KUKA KRL data list: SOLVE_HANOI.DAT

&ACCESS RVO
&REL 66
&PARAM TEMPLATE = C:\KRC\Roboter\Template\ExpertVorgabe
&PARAM EDITMASK = *
DEFDAT  SOLVE_HANOI
DECL INT I=1
DECL GLOBAL INT HANOI_DISK_COUNT=3
; Calculate REQUIRED_MOVES = 2^HANOI_DISK_COUNT - 1 (does KRL have exponents?)
DECL INT REQUIRED_MOVES=7
DECL INT MOVE_ARRAY[7,2]
DECL INT DISK_COUNTS[3]

; Remember if we come from HOME
DECL BOOL FirstMove=FALSE

; Tool Definitions
DECL GLOBAL FRAME DiskTool={x 0.0,y 0.0,z 150.0,a 0.5,b -90.5,c 0.0}

; Following are placeholders
; Info about the disk in
DECL GLOBAL REAL DISK_THICKNESS=36.65
DECL GLOBAL REAL DISK_PICKUP_OFFSET=-17

; Pick-up zone X offset
DECL GLOBAL REAL PICK_UP_X_OFFSET=-550.0

; Transit zone Z offset (currently 16" + 100mm)
DECL GLOBAL REAL TRANSIT_ZONE_Z_OFFSET=650.0

; Table coordinates for front left corner (rel to world coords)
DECL GLOBAL REAL TABLE_X=2010.0
DECL GLOBAL REAL TABLE_Y=739.775
DECL GLOBAL REAL TABLE_Z=914.4

; Towers from left to right
; Coordinate info for starting tower base relative to the table front left corner
DECL GLOBAL REAL TOWER_ONE_X=400.0
DECL GLOBAL REAL TOWER_ONE_Y=-244.1
DECL GLOBAL REAL TOWER_ONE_Z=0.0

; Coordinate info for goal tower base relative to the table front left corner
DECL GLOBAL REAL TOWER_TWO_X=400.0
DECL GLOBAL REAL TOWER_TWO_Y=-743.9
DECL GLOBAL REAL TOWER_TWO_Z=0.0

; Coordinate info for goal tower base relative to the table front left corner
DECL GLOBAL REAL TOWER_THREE_X=400.0
DECL GLOBAL REAL TOWER_THREE_Y=-1252.2
DECL GLOBAL REAL TOWER_THREE_Z=0.0
ENDDAT
